Universal Robots PolyScope program: triangle.urp

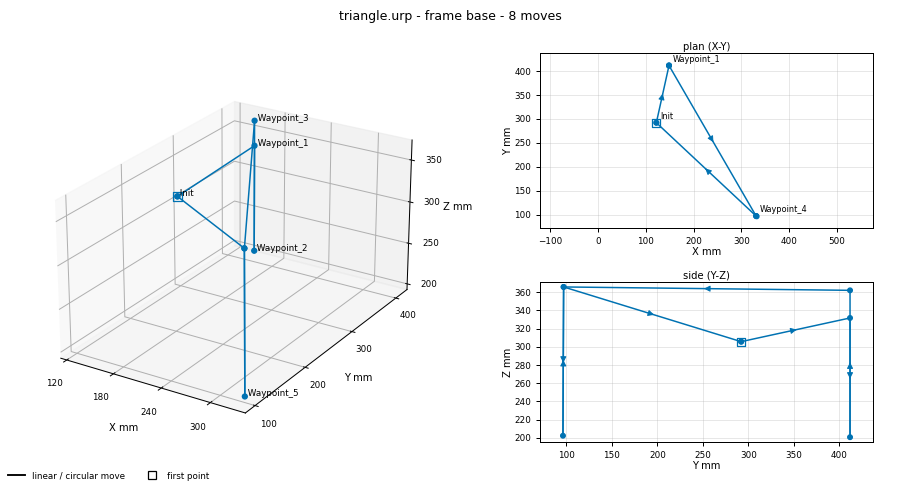
[picture p0: tool path of triangle.urp in frame base, 8 of 8 moves have a stored position in this frame; points joined in program order, loops and branches not executed]
Program triangle (installation=default directory=/programs/Mursal createdIn=5.11.11.1010533 lastSavedIn=5.11.11.1010533 robotSerialNumber=20205300864)
Calibrated DH parameters: a=[-0.000166, -0.243494, -0.153108, 0.000057, -0.000123, 0]; d=[0.151897, -1.34267, 53.988124, -52.514559, 0.085283, 0.092193]; alpha=[1.572472, -0.003756, 0.002824, 1.570807, -1.572621, 0]; deltaTheta=[0, 0.020704, 7.033215, -0.770746, 0.000004, 0]
Robot Program (runOnlyOnce=false)
  MoveL speed 250 mm/s, acceleration 1200 mm/s^2 (useActiveTCP=true) feature=Base
    Waypoint Init: TCP in base x=122.122 y=292.121 z=305.73 mm, rx=-1.1347 ry=2.9295 rz=0 rad; joints [91.64, -87.588, -91.765, -90.542, 90.031, 859.396] deg
    Waypoint Waypoint_1: TCP in base x=148.604 y=411.773 z=331.748 mm, rx=-0.8639 ry=3.015 rz=0.0164 rad; joints [87.565, -121.644, -40.964, -106.625, 89.778, 865.629] deg
    Waypoint Waypoint_2: TCP in base x=148.61 y=411.78 z=200.691 mm, rx=-0.8639 ry=3.0151 rz=0.0164 rad; joints [87.485, -121.92, -76.318, -70.997, 89.848, 865.623] deg
    URCap Gripper (Robotiq_Grippers, Robotiq Inc.) dataModel(position=100.0, force=0.0, speed=0.0, positionInDouble=100.0, forceInDouble=0.0, speedInDouble=0.0, slaveIds=[9], blocking=true, robotCompliant=false)
    Waypoint Waypoint_3: TCP in base x=148.599 y=411.783 z=362.136 mm, rx=-0.8638 ry=3.0151 rz=0.0163 rad; joints [87.607, -127.141, -22.612, -119.484, 89.73, 865.648] deg
    Waypoint Waypoint_4: TCP in base x=330.848 y=96.917 z=365.858 mm, rx=-2.7001 ry=-1.6059 rz=-0.0002 rad; joints [38.596, -97.138, -65.308, -107.444, 89.957, 967.185] deg
    Waypoint Waypoint_5: TCP in base x=331.992 y=96.209 z=202.294 mm, rx=-2.7 ry=-1.606 rz=0 rad; joints [38.289, -100.562, -106.499, -62.833, 90.025, 966.965] deg
    URCap Gripper (Robotiq_Grippers, Robotiq Inc.) dataModel(position=0.0, force=0.0, speed=0.0, positionInDouble=0.0, forceInDouble=0.0, speedInDouble=0.0, slaveIds=[9], blocking=true, robotCompliant=false)
    Waypoint Waypoint_4: TCP in base x=330.848 y=96.917 z=365.858 mm, rx=-2.7001 ry=-1.6059 rz=-0.0002 rad; joints [38.596, -97.138, -65.308, -107.444, 89.957, 967.185] deg
    Waypoint Init: TCP in base x=122.122 y=292.121 z=305.73 mm, rx=-1.1347 ry=2.9295 rz=0 rad; joints [91.64, -87.588, -91.765, -90.542, 90.031, 859.396] deg
